TYPE csp_case_feed_status_enum :
(
	CSP_CASE_FEED_STATUS_NOT_INITIALIZED 							:=  0,
	CSP_CASE_FEED_STATUS_DISABLED 									:=  10,
	CSP_CASE_FEED_STATUS_ENABLE_REQUEST 							:=  20,
	CSP_CASE_FEED_STATUS_ENABLING 									:=  30,
	CSP_CASE_FEED_STATUS_ENABLED 									:=  40,
	CSP_CASE_FEED_STATUS_CHANGE_OVER_MODE                           :=  60,
    CSP_CASE_FEED_STATUS_CHANGE_OVER_MODE_DONE                      :=  70,   
	CSP_CASE_FEED_STATUS_CALCULATING_SLAVE_POSITION					:=  90,
	CSP_CASE_FEED_STATUS_PHASE_REQUEST								:= 140,
	CSP_CASE_FEED_STATUS_PHASING									:= 150,
	CSP_CASE_FEED_STATUS_SLAVE_PHASING								:= 155,
	CSP_CASE_FEED_STATUS_CHECK_CARTON								:= 156,
	CSP_CASE_FEED_STATUS_CHECK_OK									:= 157,
	CSP_CASE_FEED_STATUS_PHASED										:= 160,
	CSP_CASE_FEED_STATUS_CAM_ENGAGED_REQ							:= 170,
	CSP_CASE_FEED_STATUS_AXIS_ENGAGE_VERIFY							:= 180,
	CSP_CASE_FEED_STATUS_CAM_ENGAGED								:= 190,
	CSP_CASE_FEED_STATUS_CAM_TABLE_READ								:= 195,
	CSP_CASE_FEED_STATUS_CALCULATE_SLAVE_POSITION_REQUEST			:= 196,
	CSP_CASE_FEED_STATUS_READY										:= 197,
	CSP_CASE_FEED_STATUS_RUNNING									:= 200,
	CSP_CASE_FEED_STATUS_MOVING										:= 205,
	CSP_CASE_FEED_STATUS_DISENGAGE_REQUEST							:= 210,
	CSP_CASE_FEED_STATUS_DISENGAGING								:= 211,			
	CSP_CASE_FEED_STATUS_DISENGAGED									:= 212,	
	CSP_CASE_FEED_STATUS_DISENGAGED_AND_STOPPED						:= 213,
	CSP_CASE_FEED_STATUS_REJECT_WAIT_FOLLOWER						:= 220,
	CSP_CASE_FEED_STATUS_REJECT_MOVE_BACK							:= 221,
	CSP_CASE_FEED_STATUS_REJECT_MOVED_BACK							:= 222,
	CSP_CASE_FEED_STATUS_REJECT_START_REJECT_SEQUENCE				:= 223,
	CSP_CASE_FEED_STATUS_REJECT_END_REJECT_SEQUENCE					:= 224,
	CSP_CASE_FEED_STATUS_REJECT_WAIT_NEW_CARTON						:= 225,
	CSP_CASE_FEED_STATUS_STOP_REQUEST 								:= 500,
	CSP_CASE_FEED_STATUS_DISABLE_REQUEST 							:= 530,
	CSP_CASE_FEED_STATUS_DISABLING 									:= 540
) := CSP_CASE_FEED_STATUS_NOT_INITIALIZED;
END_TYPE

(* stored: Version 1.1.0.1, ProductVersion 3.1.4022.12
   DUT csp_case_feed_status_enum: Id {1cc0f99a-36fe-47aa-8c0d-ef689392c19a} *)
